FUNCTION_BLOCK cylinder_2_pos
VAR_INPUT
	en_in: BOOL;
	error_bit: BOOL;
	cylinder_work_coil:BOOL;
	cylinder_home_coil:BOOL;
	delay_1: LTIME;
	delay_2: LTIME;
	
END_VAR
VAR_OUTPUT
	en_out: BOOL;
	cylinder_work_fb:BOOL;
	cylinder_home_fb:BOOL;
	delay_display_1: LTIME;
	delay_display_2: LTIME;
	
END_VAR
VAR
	sensor_delay_1: LTON;
	sensor_delay_2: LTON;
	

	
END_VAR
VAR_IN_OUT
	
END_VAR
VAR // added by the converter: edge detectors and wires of the graphical bodies
    _w1, _w2, _w3 : BOOL;
END_VAR

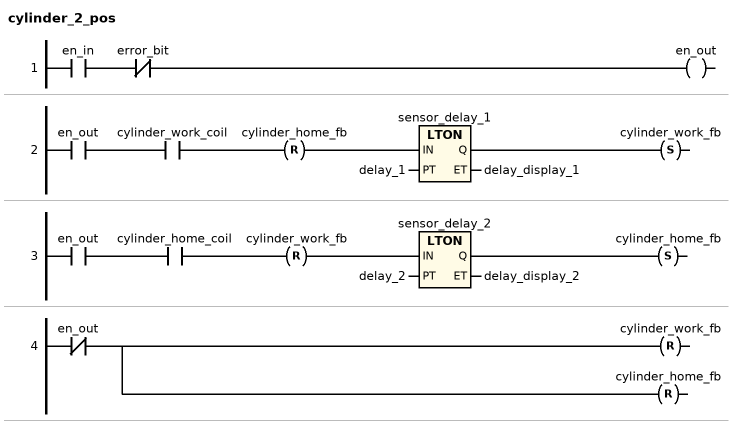
// NETWORK 1
en_out := en_in AND NOT error_bit;

// NETWORK 2
_w1 := en_out AND cylinder_work_coil;
cylinder_home_fb R= _w1;
sensor_delay_1(IN := _w1, PT := delay_1, ET => delay_display_1); // LTON
cylinder_work_fb S= sensor_delay_1.Q;

// NETWORK 3
_w2 := en_out AND cylinder_home_coil;
cylinder_work_fb R= _w2;
sensor_delay_2(IN := _w2, PT := delay_2, ET => delay_display_2); // LTON
cylinder_home_fb S= sensor_delay_2.Q;

// NETWORK 4
_w3 := NOT en_out;
cylinder_work_fb R= _w3;
cylinder_home_fb R= _w3;

END_FUNCTION_BLOCK

(* stored: Version 1.1.0.1, ProductVersion 3.1.4024.11
   POU cylinder_2_pos: Id {0cb4c0d8-b15d-49fd-88b8-ab45235b24bc}, SpecialFunc None *)
